TYPE Datalogger_SENECA :
STRUCT
	
	MesData			: Datalogger ; 			  (* (NA) MesData *)
                        			                			                            	
	MesWindSp		: REAL ;				  (* (km/h) Wind speed of the weather station on SPP zone	 		*)
	MesWindDir		: REAL ;  				  (* (deg) Wind direction of the weather station on SPP zone	    *)
	 	 						
END_STRUCT
END_TYPE

(* stored: Version 1.1.0.1, ProductVersion 3.1.4024.9
   DUT Datalogger_SENECA: Id {273a4f3f-70ba-41e7-9479-d7fbc27855ce} *)
